Staubli VAL3: load.pgx

program load()
  local num l_nResult
  local string l_sPath
begin
  // load the program  ???
  if isDefined(saveData:iInstruction[sProgType])
    call saveData:getPathInstr(sProgType,l_sPath)
    l_nResult=prog:libLoad(l_sPath)
    delay(0)
    // save the sProgTypeUsing
    saveData:sProgTypeUsing=sProgType
  endIf
end
